// TwinCAT 3 PLC project Main
// ProgramVersion: 3.1.4024.0
// libraries:
//   Tc2_Standard, * (Beckhoff Automation GmbH)
//   Tc2_System, * (Beckhoff Automation GmbH)
//   Tc2_Utilities, * (Beckhoff Automation GmbH)
//   Tc3_Module, * (Beckhoff Automation GmbH)
// project tree:
//   / PlcTask.TcTTO
//   POUs/ MAIN.TcPOU, WmicNetworkAdapterDisable.TcPOU, WmicNetworkAdapterEnable.TcPOU
// real-time tasks:
//   TASK PlcTask: cycle T#10ms, priority 20, ADS port 350

CONFIGURATION Main
    RESOURCE PLC ON TwinCAT3
        TASK PlcTask(INTERVAL := T#10ms, PRIORITY := 20);
        PROGRAM MAIN WITH PlcTask : MAIN;
    END_RESOURCE
END_CONFIGURATION

// ---- POUs/MAIN.TcPOU
PROGRAM MAIN
VAR
	enable : BOOL; // set this value true to enable
	disable : BOOL; // set this value true to disable
	wmicNetworkAdapterEnable: WmicNetworkAdapterEnable;
	wmicNetworkAdapterDisable: WmicNetworkAdapterDisable;
END_VAR

// once triggered this code will take aproximatly 10 seconds to enable or disable the adapter
// this code will work on Windows 10.  It uses Powershell and mshta, so these must be available
// on the system (which is typically already available on a Beckhoff IPC)

// when adding to your project you will need to add the Tc2_Utilities to your References.

wmicNetworkAdapterEnable(AdapterName := 'X001',Start := enable);
wmicNetworkAdapterDisable(AdapterName := 'X001',Start := disable);

IF enable AND NOT wmicNetworkAdapterEnable.Busy THEN
	enable := FALSE;
END_IF

IF disable AND NOT wmicNetworkAdapterDisable.Busy THEN
	disable := FALSE;
END_IF

END_PROGRAM

// ---- POUs/WmicNetworkAdapterEnable.TcPOU
FUNCTION_BLOCK WmicNetworkAdapterEnable
VAR_INPUT
	AdapterName : STRING(80);
    Start : BOOL;
END_VAR
VAR_OUTPUT
	Busy : BOOL;
    Error : BOOL;
    ErrorId : UDINT;
END_VAR
VAR CONSTANT
	ENABLE_CMD : T_MAXSTRING := 'C:\Windows\System32\mshta vbscript:Execute("CreateObject(""WScript.Shell"").Run ""powershell -c Enable-NetAdapter -Name """""""" -Confirm:$$false"", 0: window.close")';
	ADAPTER_INDEX_POS : INT := 124;
END_VAR
VAR
	commandLine : T_MAXSTRING;
	ntStartProcess : NT_StartProcess;
END_VAR


commandLine := INSERT(ENABLE_CMD, AdapterName, ADAPTER_INDEX_POS); 
ntStartProcess(
	NETID := '', 
	PATHSTR := commandLine, 
	DIRNAME := 'C:\Windows\System32', 
	COMNDLINE := '', 
	START := Start, 
	TMOUT := DEFAULT_ADS_TIMEOUT, 
	BUSY => Busy, 
	ERR => Error, 
	ERRID => ErrorId);

END_FUNCTION_BLOCK

// ---- POUs/WmicNetworkAdapterDisable.TcPOU
FUNCTION_BLOCK WmicNetworkAdapterDisable
VAR_INPUT
	AdapterName : STRING(80);
    Start : BOOL;
END_VAR
VAR_OUTPUT
	Busy : BOOL;
    Error : BOOL;
    ErrorId : UDINT;
END_VAR
VAR CONSTANT
	DISABLE_CMD : T_MAXSTRING := 'C:\Windows\System32\mshta vbscript:Execute("CreateObject(""WScript.Shell"").Run ""powershell -c Disable-NetAdapter -Name """""""" -Confirm:$$false"", 0: window.close")';
	ADAPTER_INDEX_POS : INT := 125;
END_VAR
VAR
	commandLine : T_MAXSTRING;
	ntStartProcess : NT_StartProcess;
END_VAR


commandLine := INSERT(DISABLE_CMD, AdapterName, ADAPTER_INDEX_POS); 
ntStartProcess(
	NETID := '', 
	PATHSTR := commandLine, 
	DIRNAME := 'C:\Windows\System32', 
	COMNDLINE := '', 
	START := Start, 
	TMOUT := DEFAULT_ADS_TIMEOUT, 
	BUSY => Busy, 
	ERR => Error, 
	ERRID => ErrorId);

END_FUNCTION_BLOCK
